TYPE Tank_Io_Out :
STRUCT
	bInletValveOpen		: BOOL;
END_STRUCT
END_TYPE

(* stored: Version 1.1.0.1
   DUT Tank_Io_Out: Id {f548bb91-b729-4956-a1c3-c2096a52c9f9} *)
